TYPE ST_UTILITY :
STRUCT
	TOTAL_FLOW_CAL:DINT;
	TOTAL_FLOW_MO:DINT;
	SPARE_1:DINT;
	SPARE_2:DINT;
	SPARE_3:DINT;
	SPARE_4:DINT;
	SPARE_5:DINT;
	SPARE_6:DINT;
	SPARE_7:DINT;
	SPARE_8:DINT;
	SPARE_9:DINT;
	SPARE_10:DINT;
END_STRUCT
END_TYPE

(* stored: Version 1.1.0.1, ProductVersion 3.1.4024.12
   DUT ST_UTILITY: Id {20f1ecec-1dc6-4727-9841-30df89d490e8} *)
